// TIA Portal project "Process control system" (V17)

(* hardware
DEVICE "S7-1200 station_1"  S7-1200 Station
   slot 0: "Rack_0"  S7-1200 Rack  Rack  V1.0
   slot 1: "PLC_1"  CPU 1212C DC/DC/DC  6ES7 212-1AE40-0XB0  V4.2
   slot 2: "AI 4x13BIT/AQ 2x14BIT_1"  6ES7 234-4HE32-0XB0  V2.1
*)

// ===== PLC "PLC_1"  CPU 1212C DC/DC/DC =====

VAR_GLOBAL   // PLC tag table "Default tag table"
   "levelSensor1" AT %IW96 : Int;
   "flowValve" AT %QW96 : Int;
END_VAR

VAR_GLOBAL   // PLC tag table "PLCTags"
   "Start_SS1" AT %I0.0 : Bool;
   "Stop_SS2" AT %I0.1 : Bool;
   "SV1" AT %Q0.1 : Bool;
   "Pump" AT %Q0.0 : Bool;
   "SV2" AT %Q0.3 : Bool;
END_VAR

DATA_BLOCK "ourDataBlock"   // DB2
{ S7_Optimized_Access := 'TRUE' }
VERSION : 0.1
   VAR
      levelSensorVal : Int;
      levelSensorMin : Int := 4085;
      levelSensorMax : Int := 13928;
      normXOut : Real;
      tankWaterLevel : Real;
   END_VAR
BEGIN
END_DATA_BLOCK

FUNCTION "normXScaleX" : Void   // FC1, LAD
{ S7_Optimized_Access := 'TRUE' }
VERSION : 0.1
BEGIN

REGION Network 1: NormX
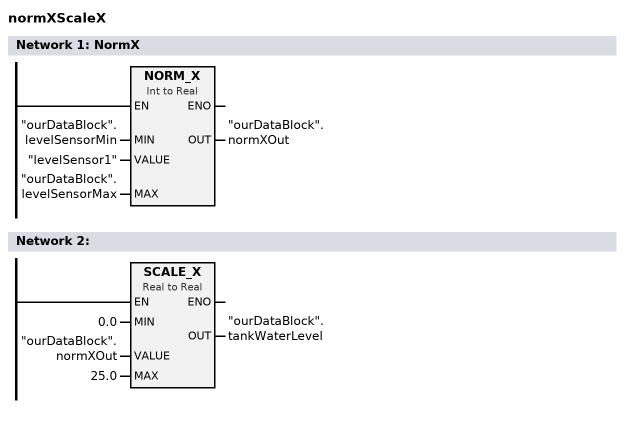
   RUNG wire#powerrail
      { S7_Templates := "[SrcType := Int, DestType := Real]" } Normalize(min := "ourDataBlock".levelSensorMin, value := "levelSensor1", max := "ourDataBlock".levelSensorMax, out => "ourDataBlock".normXOut)
   END_RUNG
   // the same network as SCL:
   "ourDataBlock".normXOut := NORM_X(MIN := "ourDataBlock".levelSensorMin, VALUE := "levelSensor1", MAX := "ourDataBlock".levelSensorMax);
END_REGION

REGION Network 2
   RUNG wire#powerrail
      { S7_Templates := "[SrcType := Real, DestType := Real]" } Scale(min := 0.0, value := "ourDataBlock".normXOut, max := 25.0, out => "ourDataBlock".tankWaterLevel)
   END_RUNG
   // the same network as SCL:
   "ourDataBlock".tankWaterLevel := SCALE_X(MIN := 0.0, VALUE := "ourDataBlock".normXOut, MAX := 25.0);
END_REGION
END_FUNCTION

FUNCTION "FillingProcess" : Void   // FC2, LAD
{ S7_Optimized_Access := 'TRUE' }
VERSION : 0.1
BEGIN

REGION Network 1
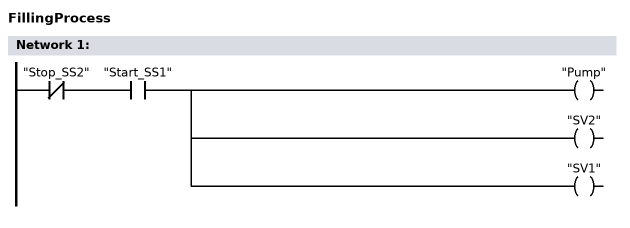
   RUNG wire#powerrail
      I_Contact( "Stop_SS2" )
      Contact( "Start_SS1" )
      wire#w1
      Coil( "Pump" )
   END_RUNG
   RUNG wire#w1
      Coil( "SV2" )
   END_RUNG
   RUNG wire#w1
      Coil( "SV1" )
   END_RUNG
   // the same network as SCL:
   "Pump" := NOT "Stop_SS2" AND "Start_SS1";
   "SV2" := "Pump";
   "SV1" := "Pump";
END_REGION
END_FUNCTION

ORGANIZATION_BLOCK "Main"   // OB1, LAD, ProgramCycle
TITLE = "Main Program Sweep (Cycle)"
{ S7_Optimized_Access := 'TRUE' }
VERSION : 0.1
   VAR_INPUT
      Initial_Call : Bool;   // Initial call of this OB
      Remanence : Bool;   // =True, if remanent data are available
   END_VAR
BEGIN

REGION Network 1
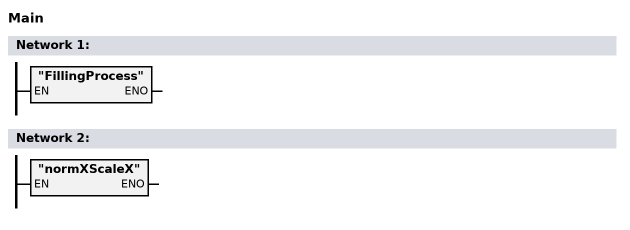
   RUNG wire#powerrail
      "FillingProcess"()
   END_RUNG
   // the same network as SCL:
   "FillingProcess"();
END_REGION

REGION Network 2
   RUNG wire#powerrail
      "normXScaleX"()
   END_RUNG
   // the same network as SCL:
   "normXScaleX"();
END_REGION
END_ORGANIZATION_BLOCK

ORGANIZATION_BLOCK "PIDControlller"   // OB30, LAD, CyclicInterrupt
{ S7_Optimized_Access := 'TRUE' }
VERSION : 0.1
   VAR_INPUT
      Initial_Call : Bool;   // Initial call of this OB
      Event_Count : Int;   // Events discarded
   END_VAR
BEGIN

REGION Network 1: Inserting the PID compact block
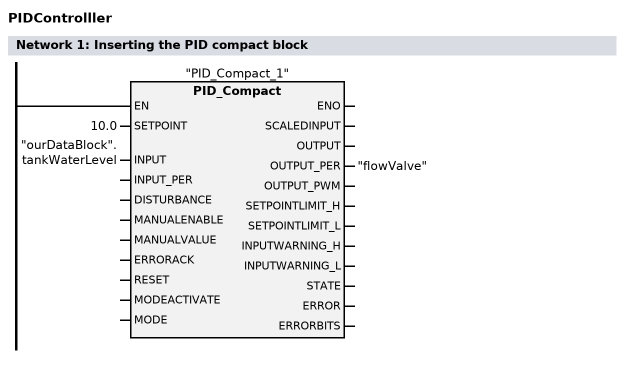
   "PID_Compact_1"(Setpoint := 10.0, Input := "ourDataBlock".tankWaterLevel, Output_PER => "flowValve");   // PID_Compact
END_REGION
END_ORGANIZATION_BLOCK